{attribute 'qualified_only'}
{attribute 'strict'}
TYPE E_Huawei_SmartLogger_Error_1 :
(
	eNoError := 0,
	eModbusTCPError := 1,
	eHuawei_SmartLoggerError := 2,
	eHuawei_SmartLoggerTooBigValueReceived := 3
);
END_TYPE

(* stored: Version 1.1.0.1, ProductVersion 3.1.4024.11
   DUT E_Huawei_SmartLogger_Error_1: Id {22d94502-5af3-4a4b-b1fe-cf90f5cf4ad7} *)
